(* CODESYS project Clock.xml

Project tree, tasks and I/O mapping:
  program Clock [LD]
*)

// Clock
PROGRAM Clock
VAR
	Timezone: TimezoneInformation;
END_VAR

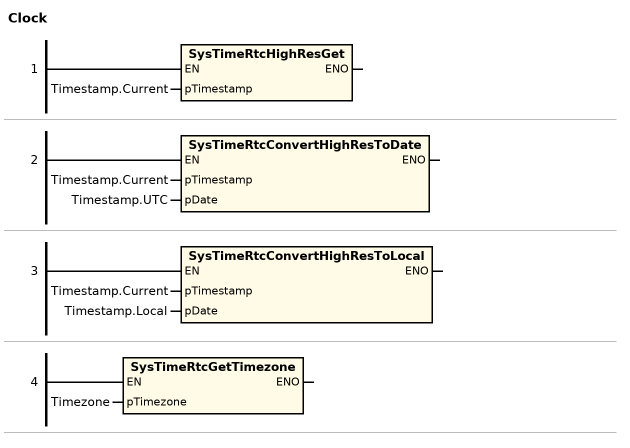
// NETWORK 1
SysTimeRtcHighResGet(pTimestamp := Timestamp.Current);

// NETWORK 2
SysTimeRtcConvertHighResToDate(pTimestamp := Timestamp.Current, pDate := Timestamp.UTC);

// NETWORK 3
SysTimeRtcConvertHighResToLocal(pTimestamp := Timestamp.Current, pDate := Timestamp.Local);

// NETWORK 4
SysTimeRtcGetTimezone(pTimezone := Timezone);

END_PROGRAM
